// TIA Portal V19 export
TYPE "LEXCHANGETRAY_typePc_controlNode"
// stored: Access Published
   STRUCT
      cmd { S7_SetPoint := 'True'} : "LEXCHANGETRAY_typePc_Cmd";   // Command for control node
      par { S7_SetPoint := 'True'} : "LEXCHANGETRAY_typePc_controlPar";   // Control parameters
      monitor { S7_SetPoint := 'True'} : "LEXCHANGETRAY_typePc_Monitor";   // Tray status / 托盘状态
   END_STRUCT;
END_TYPE
